PROGRAM MAIN
VAR
    motor : FB_Motor;
END_VAR

motor.SetSpeed(value := 1.0);
motor.Stop();

END_PROGRAM

(* stored: Version 1.1.0.1, ProductVersion 3.1.4024.0
   POU MAIN: Id {9a3f04d7-2e6b-4c81-b5a0-73f18d92c6e4}, SpecialFunc None *)
